// TwinCAT 3 PLC project ProfilerTest
// ProgramVersion: 3.1.4024.0
// libraries:
//   Tc2_Standard, * (Beckhoff Automation GmbH)
//   Tc2_System, * (Beckhoff Automation GmbH)
//   Tc2_Utilities, * (Beckhoff Automation GmbH)
//   Tc3_Module, * (Beckhoff Automation GmbH)
// project tree:
//   / PlcTask.TcTTO
//   POUs/ Factorial.TcPOU (not stored), MAIN.TcPOU
// (motion and I/O tree: see PLC project buffertest)
// real-time tasks:
//   TASK PlcTask: cycle T#10ms, priority 20, ADS port 350
//   TASK PlcTask1: cycle T#10ms, priority 21, ADS port 351

CONFIGURATION ProfilerTest
    RESOURCE PLC ON TwinCAT3
        TASK PlcTask(INTERVAL := T#10ms, PRIORITY := 21);
        PROGRAM MAIN WITH PlcTask : MAIN;
    END_RESOURCE
END_CONFIGURATION

// ---- POUs/MAIN.TcPOU
PROGRAM MAIN
VAR
	nFactorial : ULINT;
	Profiler : PROFILER;
	ProfilerResult : PROFILERSTRUCT;
END_VAR

Profiler(START := TRUE, RESET := FALSE);
Factorial(n := nFactorial);
Profiler(START := FALSE);
ProfilerResult := Profiler.DATA;

END_PROGRAM
